{attribute 'qualified_only'}
VAR_GLOBAL



	
	
END_VAR

(* stored: Version 1.1.0.1, ProductVersion 3.1.4024.0
   GVL GVL: Id {73215583-16c3-464d-b4af-a91b5af9be94} *)
